	DATA_BLOCK DB295
	TITLE =DBG195M  INLET SLIDE GERM 5
	//COPYRIGHT:    (C) 2009  BUHLER AG, CH-9240 UZWIL, SWITZERLAND
	//
	//PRODUCT:      WinCoS_BIW01_09
	//
	//TITLE:        INLET SLIDE GERM 5
	//                Machine group DB
	//                Maschinengruppen-DB
	//
	//-------------------------------------------------------------------------
	//
	//IDENT:        AUTHOR:             DEPT:             DATE:
	//
	//P01_DB295.1.0 K.Renz              CSB41             13.Jan.2010
	//              1st Release
	//
	//-------------------------------------------------------------------------
	//
	//PURPOSE:
	//
	//MANUAL :
	//
	//RESTRICTIONS:
	//
	//-------------------------------------------------------------------------
	AUTHOR  : KR
	FAMILY  : USW
	NAME    : DBG195M
	VERSION : 00.00

	FB295
	BEGIN
	      #Gr.Par.ParObjectNo 	:=19500;
	      #Gr.Par.ParIdling      	:=2;
	      #Gr.Par.ParMgr	        :=True;
	      #Gr.Par.ParWgr	        :=False;
	      #Gr.Par.ParGgr	        :=False;
	      #Gr.Par.ParEmptyingTime 	:=0;
	      #Gr.Par.ParHornCode       :=6;
	//Parameter =A-2502-BZS13 : DISCHARGE CHUTE PARKING POSITION
	      #A_2502_BZS13.Par.ParObjectNo                             :=19501;
	      #A_2502_BZS13.Par.ParMsgType                              :=7163;
	      #A_2502_BZS13.Par.ParHornCode                             :=6;
	      #A_2502_BZS13.Par.ParDelayChange                          :=20;
	      #A_2502_BZS13.Par.ParDelayTrue                            :=10;
	      #A_2502_BZS13.Par.ParDelayFalse                           :=0;
	      #A_2502_BZS13.Par.ParTimeoutTrue                          :=0;
	      #A_2502_BZS13.Par.ParTimeoutFalse                         :=0;
	      #A_2502_BZS13.Par.ParLogOff                               :=False;
	      #A_2502_BZS13.Par.Par2WorkingCond                         :=False;
	      #A_2502_BZS13.Par.ParFaultRetry                           :=False;
	      #A_2502_BZS13.Par.ParBinLevel                             :=False;
	//
	//
	//Parameter =A-2502-BZS14 : DISCHARGE CHUTE LEFT SIDE
	      #A_2502_BZS14.Par.ParObjectNo                             :=19502;
	      #A_2502_BZS14.Par.ParMsgType                              :=7163;
	      #A_2502_BZS14.Par.ParHornCode                             :=6;
	      #A_2502_BZS14.Par.ParDelayChange                          :=20;
	      #A_2502_BZS14.Par.ParDelayTrue                            :=10;
	      #A_2502_BZS14.Par.ParDelayFalse                           :=0;
	      #A_2502_BZS14.Par.ParTimeoutTrue                          :=0;
	      #A_2502_BZS14.Par.ParTimeoutFalse                         :=0;
	      #A_2502_BZS14.Par.ParLogOff                               :=False;
	      #A_2502_BZS14.Par.Par2WorkingCond                         :=False;
	      #A_2502_BZS14.Par.ParFaultRetry                           :=False;
	      #A_2502_BZS14.Par.ParBinLevel                             :=False;
	//
	//
	//Parameter =A-2502-BZS15 : DISCHARGE CHUTE RIGHT SIDE
	      #A_2502_BZS15.Par.ParObjectNo                             :=19503;
	      #A_2502_BZS15.Par.ParMsgType                              :=7163;
	      #A_2502_BZS15.Par.ParHornCode                             :=6;
	      #A_2502_BZS15.Par.ParDelayChange                          :=20;
	      #A_2502_BZS15.Par.ParDelayTrue                            :=10;
	      #A_2502_BZS15.Par.ParDelayFalse                           :=0;
	      #A_2502_BZS15.Par.ParTimeoutTrue                          :=0;
	      #A_2502_BZS15.Par.ParTimeoutFalse                         :=0;
	      #A_2502_BZS15.Par.ParLogOff                               :=False;
	      #A_2502_BZS15.Par.Par2WorkingCond                         :=False;
	      #A_2502_BZS15.Par.ParFaultRetry                           :=False;
	      #A_2502_BZS15.Par.ParBinLevel                             :=False;
	//
	//
	//Parameter =A-2502-MXZ01 : CHUTE DRIVE
	      #A_2502_MXZ01.Par.ParObjectNo                             :=19504;
	      #A_2502_MXZ01.Par.ParMsgType                              :=7056;
	      #A_2502_MXZ01.Par.ParHornCode                             :=6;
	      #A_2502_MXZ01.Par.ParMonTime                              :=20;
	      #A_2502_MXZ01.Par.ParStartingTime                         :=20;
	      #A_2502_MXZ01.Par.ParStoppingTime                         :=50;
	      #A_2502_MXZ01.Par.ParIdlingTime                           :=0;
	      #A_2502_MXZ01.Par.ParDelayTime                            :=10;
	      #A_2502_MXZ01.Par.ParLogOff                               :=False;
	      #A_2502_MXZ01.Par.ParManual                               :=True;
	      #A_2502_MXZ01.Par.ParRestartDelay                         :=False;
	      #A_2502_MXZ01.Par.Par2Speed                               :=False;
	      #A_2502_MXZ01.Par.ParHeavyStartup                         :=False;
	//
	//
	//Parameter =A-2502-QYS21 : DISCHARGE CHUTE LEFT SIDE
	      #A_2502_QYS21.Par.ParObjectNo                             :=19505;
	      #A_2502_QYS21.Par.ParMsgType                              :=7163;
	      #A_2502_QYS21.Par.ParHornCode                             :=6;
	      #A_2502_QYS21.Par.ParDelayChange                          :=20;
	      #A_2502_QYS21.Par.ParDelayTrue                            :=10;
	      #A_2502_QYS21.Par.ParDelayFalse                           :=0;
	      #A_2502_QYS21.Par.ParTimeoutTrue                          :=0;
	      #A_2502_QYS21.Par.ParTimeoutFalse                         :=0;
	      #A_2502_QYS21.Par.ParLogOff                               :=False;
	      #A_2502_QYS21.Par.Par2WorkingCond                         :=False;
	      #A_2502_QYS21.Par.ParFaultRetry                           :=False;
	      #A_2502_QYS21.Par.ParBinLevel                             :=False;
	//
	//
	//Parameter =A-2502-QYS22 : DISCHARGE CHUTE RIGHT SIDE
	      #A_2502_QYS22.Par.ParObjectNo                             :=19506;
	      #A_2502_QYS22.Par.ParMsgType                              :=7163;
	      #A_2502_QYS22.Par.ParHornCode                             :=6;
	      #A_2502_QYS22.Par.ParDelayChange                          :=20;
	      #A_2502_QYS22.Par.ParDelayTrue                            :=10;
	      #A_2502_QYS22.Par.ParDelayFalse                           :=0;
	      #A_2502_QYS22.Par.ParTimeoutTrue                          :=0;
	      #A_2502_QYS22.Par.ParTimeoutFalse                         :=0;
	      #A_2502_QYS22.Par.ParLogOff                               :=False;
	      #A_2502_QYS22.Par.Par2WorkingCond                         :=False;
	      #A_2502_QYS22.Par.ParFaultRetry                           :=False;
	      #A_2502_QYS22.Par.ParBinLevel                             :=False;
	//
	//
	END_DATA_BLOCK
